// TIA Portal V18 export
FUNCTION "Enable-Axis" : Void   // FC3, LAD
{ S7_Optimized_Access := 'TRUE' }
AUTHOR : HenriP
VERSION : 0.1
// stored: AutoNumber true, IsIECCheckEnabled false, SetENOAutomatically false, UDAEnableTagReadback false
   VAR_INPUT
      Enable : Bool;
      "E-STOP" : Bool;
      Stop : Bool;
      Halt : Bool;
   END_VAR
   VAR_OUTPUT
      FestoStop : Bool;
      FestoEnable : Bool;
      FestoHalt : Bool;
   END_VAR
BEGIN

REGION Network 1: Festo Enable
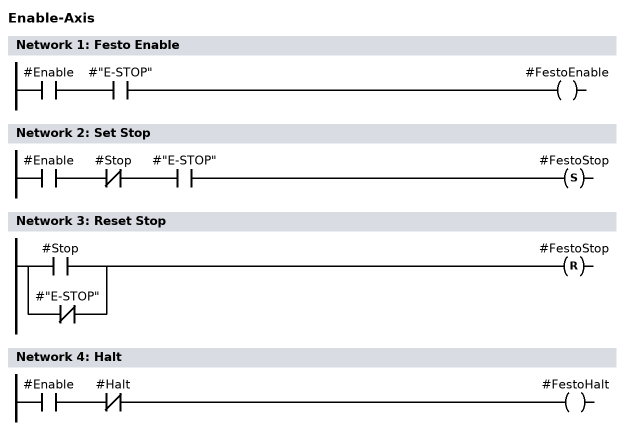
   RUNG wire#powerrail
      Contact( #Enable )
      Contact( #"E-STOP" )
      Coil( #FestoEnable )
   END_RUNG
   // the same network as SCL:
   #FestoEnable := #Enable AND #"E-STOP";
END_REGION

REGION Network 2: Set Stop
   RUNG wire#powerrail
      Contact( #Enable )
      I_Contact( #Stop )
      Contact( #"E-STOP" )
      S_Coil( #FestoStop )
   END_RUNG
   // the same network as SCL:
   IF #Enable AND NOT #Stop AND #"E-STOP" THEN #FestoStop := TRUE; END_IF;
END_REGION

REGION Network 3: Reset Stop
   RUNG wire#powerrail
      Contact( #Stop )
      wire#w1
      R_Coil( #FestoStop )
   END_RUNG
   RUNG wire#powerrail
      I_Contact( #"E-STOP" )
   END_RUNG wire#w1
   // the same network as SCL:
   IF #Stop OR NOT #"E-STOP" THEN #FestoStop := FALSE; END_IF;
END_REGION

REGION Network 4: Halt
   RUNG wire#powerrail
      Contact( #Enable )
      I_Contact( #Halt )
      Coil( #FestoHalt )
   END_RUNG
   // the same network as SCL:
   #FestoHalt := #Enable AND NOT #Halt;
END_REGION
END_FUNCTION
